// TIA Portal V19 export
DATA_BLOCK "LB101"   // DB86
// stored: InstanceOfName ButtonsSafe_LB101, InstanceOfType FB
"ButtonsSafe_LB101"
   // VAR_INPUT
   //    Reset_OthersPBs_Activation_IN : Bool;
   // END_VAR
   // VAR_OUTPUT
   //    Reset_OthersPBs_Activation_OUT : Bool;
   // END_VAR
   // VAR
   //    i : Int;
   //    iOperation : Int;
   //    iConcurrentOperation : Int;
   //    SettingWriteDone { S7_SetPoint := 'True'} : Bool;
   //    PbPanel { S7_SetPoint := 'True'} : "Buttons2Hands";
   //    PB : Struct
   //       ResetAlarms : Bool;
   //       Decoiler1InLine : Bool;
   //       Decoiler2InLine : Bool;
   //    END_STRUCT;
   // END_VAR
BEGIN
END_DATA_BLOCK
